FUNCTION F_AnyToString : STRING(255)
VAR_INPUT
		Value:		ANY;
END_VAR
VAR
    pSINT:		POINTER TO SINT;
    pUSINT:		POINTER TO USINT;
    pWORD:		POINTER TO WORD;//16 bit
    pINT:		POINTER TO INT; //16 bit
    pUINT:		POINTER TO UINT; //16 bit
	
    pDINT:		POINTER TO DINT; //32 bit
    pUDINT:		POINTER TO UDINT; //32 bit
    pDWORD:		POINTER TO DWORD; //32 bit
    pREAL:		POINTER TO REAL; //32 bit
	
    pLREAL:		POINTER TO LREAL; //64 bit
    pLWORD:		POINTER TO LWORD; //64 bit
    
END_VAR

CASE Value.TypeClass OF
// BYTE
	__SYSTEM.TYPE_CLASS.TYPE_BYTE:
		F_AnyToString:= BYTE_TO_STRING(Value.pValue^);
// SINT
	__SYSTEM.TYPE_CLASS.TYPE_SINT:
		pSINT:= Value.pValue;
		F_AnyToString:= SINT_TO_STRING(pSINT^);
// USINT
    __SYSTEM.TYPE_CLASS.TYPE_USINT:
		pUSINT:= Value.pValue;
		F_AnyToString:= USINT_TO_STRING(pUSINT^);
// WORD
    __SYSTEM.TYPE_CLASS.TYPE_WORD:
		pWORD:= Value.pValue;
		F_AnyToString:= WORD_TO_STRING(pWORD^);
// INT
    __SYSTEM.TYPE_CLASS.TYPE_INT:
		pINT:= Value.pValue;
		F_AnyToString:= INT_TO_STRING(pINT^);
// UINT
    __SYSTEM.TYPE_CLASS.TYPE_UINT:
		pUINT:= Value.pValue;
		F_AnyToString:= UINT_TO_STRING(pUINT^);
// DINT
    __SYSTEM.TYPE_CLASS.TYPE_DINT:
		pDINT:= Value.pValue;
		F_AnyToString:= DINT_TO_STRING(pDINT^);
// UDINT
    __SYSTEM.TYPE_CLASS.TYPE_UDINT:
		pUDINT:= Value.pValue;
		F_AnyToString:= UDINT_TO_STRING(pUDINT^);
// DWORD
    __SYSTEM.TYPE_CLASS.TYPE_DWORD:
		pDWORD:= Value.pValue;
		F_AnyToString:= DWORD_TO_STRING(pDWORD^); 
// REAL
    __SYSTEM.TYPE_CLASS.TYPE_REAL:
		pREAL:= Value.pValue;
		F_AnyToString:= REAL_TO_STRING(pREAL^);
// LREAL
    __SYSTEM.TYPE_CLASS.TYPE_LREAL:
		pLREAL:= Value.pValue;
		F_AnyToString:= LREAL_TO_STRING(pLREAL^);

 	
END_CASE

END_FUNCTION

(* stored: Version 1.1.0.1
   POU F_AnyToString: Id {c83ec4cb-bcaf-08af-3d29-8e246087fb4f}, SpecialFunc None *)
